TYPE IOTypes :
STRUCT
	DIn: DigitalInputs;
	DOut: DigitalOutputs;
	AIn: AnalogInputs;
	AOut: AnalogOutputs;
	ModbusRTU: ModbusRTU_IO; 
END_STRUCT
END_TYPE

(* stored: Version 1.1.0.1, ProductVersion 3.1.4024.6
   DUT IOTypes: Id {53f9b43a-b471-4210-b092-9233fb18c923} *)
